TYPE ST_KBUS_KL1501DataIn :
STRUCT
	nState	: BYTE;
	arrData	: ARRAY [0..1] OF UINT;
END_STRUCT
END_TYPE

(* stored: Version 1.1.0.1, ProductVersion 3.1.4024.15
   DUT ST_KBUS_KL1501DataIn: Id {6a6e3943-6585-4d11-88da-9d2c4256aede} *)
